PROGRAM MAIN
VAR
	TP0: FB_Torque_prediction;
END_VAR

TP0();

END_PROGRAM

(* stored: Version 1.1.0.1, ProductVersion 3.1.4024.0
   POU MAIN: Id {669ec0ec-14f4-4f97-93d0-387805f25cf8}, SpecialFunc None *)
